Staubli VAL3: onInsert.pgx

public program onInsert(string& x_sItem[])
  local string l_sItem
begin
  //
  // compose the string
  // call getType(l_sItem)
  // x_sItem=l_sItem+" ???"
  //
end
